// TIA Portal V15.1 export
// export: Created 2026-01-09T13:45:16.0514812Z, ExportSetting WithDefaults, WithReadOnly, DisplayName Totally Integrated Automation Portal, DisplayVersion V15.1 Update 8, DisplayName TIA Portal Openness, DisplayVersion V15.1 Update 8, DisplayName STEP 7 Professional, DisplayVersion V15.1 Update 8, DisplayName WinCC Advanced, DisplayVersion V15.1 Update 8
DATA_BLOCK "9.4.DLC_ADD3"   // DB916
{ S7_Optimized_Access := 'TRUE' }
VERSION : 0.1
// stored: AutoNumber true, CodeModifiedDate 2025-08-27T17:14:35.2407356Z, CompileDate 2025-08-30T17:40:35.4487891Z, CreationDate 2024-10-14T17:30:23.9104835Z, DBAccessibleFromOPCUA true, DownloadWithoutReinit false, InstanceOfName 9.TIMER_DELAY, InstanceOfNumber 9, InstanceOfType FB, InterfaceModifiedDate 2022-05-24T16:36:11.1705081Z, IsConsistent true, IsKnowHowProtected false, IsRetainMemResEnabled false, MemoryReserve 100, ModifiedDate 2025-08-27T17:14:35.2407356Z, ParameterModified 2022-05-24T16:36:11.1705081Z, StructureModified 2022-05-24T16:36:11.1705081Z, UDAEnableTagReadback false
"9.TIMER_DELAY"
   // VAR_INPUT
   //    ON : Bool;
   //    CLOCK_1S : Bool;
   //    T_DELAY : Real;
   // END_VAR
   // VAR_OUTPUT
   //    OUT : Bool;
   //    T_OUT : Real;
   // END_VAR
   // VAR
   //    TDL : Real;
   //    CLK : Bool;
   // END_VAR
BEGIN
END_DATA_BLOCK
